# B&R Automation Studio project PloterCNC
Automation Studio 4.7.5.60 SP; technology packages: mapp 5.14.1, mappCockpit 5.14.0, mappMotion 5.14.2, mappView 5.14.2

## Configuration Config1

CPU X20CP1684, AutomationRuntime D4.73, Build 4.1.2, Safety 0.0, Vc V4.72.0

### Task classes (Cpu.sw)
```
Cyclic#1 (cycle 4000 us, tolerance 0 us):
  Initiation <- Programs.CNC_Programs.InitiationandHoming.prg
  ManualCont <- Programs.CNC_Programs.ManualContr.prg
  RuchZGCode <- Programs.CNC_Programs.RuchZGCode.prg
  live_draw <- Programs.live_drawing.live_draw.prg
Cyclic#3 (cycle 48000 us, tolerance 48000 us):
  UsrMgmtP <- Programs.UsrMgmtP.prg
Cyclic#4:
  svg_to_gco <- Programs.live_drawing.svg_to_gcode.prg
  Alarm <- Programs.Alarm.prg
Cyclic#8 (cycle 8000 us, tolerance 32000 us):
  Recipe <- Programs.Recipe.prg
DataObjects: McAcpSys
NcDataObjects: InitCncPro
Binaries: udbdef, arsvcreg, FWRules, McAcpDrv, McMechSys, mvLoader, McAcpSim, TCData, arflatprv, arcoal, TCLang, mCoWebSc, iomap, Config_4, asfw, Config_3, Role, ashwd, User, Config_1, Config_2, arconfig, Hierarchy, sysconf, ashwac, Config_6, UsrMgmt, UsrLog, TC, AlarmGnrl, Recipe_cfg, GroupGlobl, GroupFile, AlarmGlobl, GroupCnc, AlarmCnc, GroupGnrl, History, AlarmFile, Settings, Config_5, Config
Libraries: McBase, MpCnc, McAxGroup, McPathGen, McAxis, McProgInt, McAcpAx, MpAlarmX, astime, runtime, MpUserX, FileIO, MpFile, MpServer, asstring, CoTrace, AsZip, MpCom, MpBase, standard, MpWebXs, AsArSdm, MpAxis, AsBrStr, MpRecipe, sys_lib, arcert, aseth, ashw, arssl, powerlnk, asieccon, asmem, asarprof, dataobj, brsystem, asarlog, aruser, asusb, asepl, MpTweet
```

### Hardware
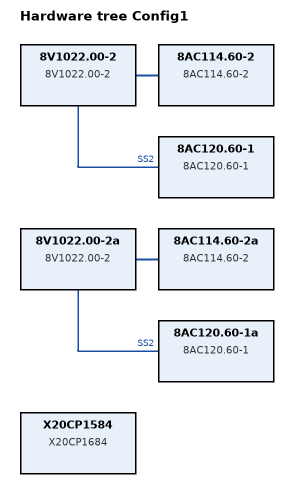
```
8AC114.60-2 : 8AC114.60-2 v1.0.0.8  [SS -> 8V1022.00-2.SS1; PLK2 -> 8AC114.60-2a.PLK2 [Cable Type=PowerlinkCable, Length=10, Version=1.0.0.2]]
8AC114.60-2a : 8AC114.60-2 v1.0.0.8  [SS -> 8V1022.00-2a.SS1; PLK1 -> X20CP1584.IF3 [Cable Type=PowerlinkCable, Length=10, Version=1.0.0.2]; PLK2 -> 8AC114.60-2.PLK2 [Cable Type=PowerlinkCable, Length=10, Version=1.0.0.2]]
8AC120.60-1 : 8AC120.60-1 v2.2.0.0  [SS -> 8V1022.00-2.SS2]
  PlugInType = Encoder
  McAcoposTypeID = AcoposPlugInConfig
8AC120.60-1a : 8AC120.60-1 v2.2.0.0  [SS -> 8V1022.00-2a.SS2]
  PlugInType = Encoder
  McAcoposTypeID = AcoposPlugInConfig
8V1022.00-2 : 8V1022.00-2 v2.2.0.0
  DriveConfiguration/Module:
    McAcoposTypeID = AcoposConfig
    ActivateACOPOSSimulationOnPLC = 0
  DriveConfiguration/Channel[1]/RealAxis:
    AxisReference = gAxisQZ
  DriveConfiguration/Channel[1]/RealAxis/MechanicalElements/Gearbox:
    InputIsReadOnly = 0
    Input = 1
    OutputIsReadOnly = 0
    Output = 1
  DriveConfiguration/Channel[1]/RealAxis/MechanicalElements/RotaryToLinearTransformation:
    ReferenceDistanceIsReadOnly = 0
    ReferenceDistance = 1.385
  DriveConfiguration/Channel[1]/RealAxis/Controller:
    ModeIsReadOnly = 0
    Mode = PositionController
  DriveConfiguration/Channel[1]/RealAxis/Controller/Mode/Position:
    ProportionalGain = 540.999939
    IntegrationTime = 0.0
    PredictionTime = 0.0004
    TotalDelayTime = 0.0004
  DriveConfiguration/Channel[1]/RealAxis/Controller/Mode/Speed:
    ProportionalGainIsReadOnly = 0
    ProportionalGain = 0.950000
    IntegrationTimeIsReadOnly = 0
    IntegrationTime = 0.0
    FilterTimeIsReadOnly = 0
    FilterTime = 0.0
  DriveConfiguration/Channel[1]/RealAxis/Controller/Mode/LoopFilters:
    LoopFilter1 = NotUsed
    LoopFilter2 = NotUsed
    LoopFilter3 = NotUsed
  DriveConfiguration/Channel[1]/RealAxis/Homing:
    Mode = Absolute
  DriveConfiguration/Channel[1]/RealAxis/Homing/Mode:
    Position = -1352
  DriveConfiguration/Channel[1]/RealAxis/Homing:
    RestorePositionVariable = 
  DriveConfiguration/Channel[1]/RealAxis/StopReaction:
    Quickstop = DecelerationLimit
    DriveError = DecelerationLimit
  DriveConfiguration/Channel[1]/RealAxis/MovementErrorLimits:
    PositionError = 1.0
    VelocityErrorMonitoring = Automatic1
  DriveConfiguration/Channel[1]/RealAxis:
    JerkFilter = NotUsed
  DriveConfiguration/Channel[1]/RealAxis/DigitalInputs/HomingSwitch:
    Level = High
  DriveConfiguration/Channel[1]/RealAxis/DigitalInputs/PositiveLimitSwitch:
    Level = Low
  DriveConfiguration/Channel[1]/RealAxis/DigitalInputs/NegativeLimitSwitch:
    Level = Low
  DriveConfiguration/Channel[1]/RealAxis/DigitalInputs/Trigger1:
    Level = High
  DriveConfiguration/Channel[1]/RealAxis/DigitalInputs/Trigger2:
    Level = High
  DriveConfiguration/Channel[1]/RealAxis/DigitalInputs/Quickstop:
    Input = Trigger2
  DriveConfiguration/Channel[1]/RealAxis/Simulation:
    SimulationModeOnPLC = SetValueGeneration
    SimulationModeOnACOPOS = NotUsed
8V1022.00-2a : 8V1022.00-2 v2.2.0.0
  DriveConfiguration/Module:
    McAcoposTypeID = AcoposConfig
    ActivateACOPOSSimulationOnPLC = 0
  DriveConfiguration/Channel[1]/RealAxis:
    AxisReference = gAxisQX
  DriveConfiguration/Channel[1]/RealAxis/MechanicalElements/Gearbox:
    InputIsReadOnly = 0
    Input = 1
    OutputIsReadOnly = 0
    Output = 1
  DriveConfiguration/Channel[1]/RealAxis/MechanicalElements/RotaryToLinearTransformation:
    ReferenceDistanceIsReadOnly = 0
    ReferenceDistance = 1.385
  DriveConfiguration/Channel[1]/RealAxis/Controller:
    ModeIsReadOnly = 0
    Mode = PositionController
  DriveConfiguration/Channel[1]/RealAxis/Controller/Mode/Position:
    ProportionalGain = 398.999969
    IntegrationTime = 0.0
    PredictionTime = 0.0004
    TotalDelayTime = 0.0004
  DriveConfiguration/Channel[1]/RealAxis/Controller/Mode/Speed:
    ProportionalGainIsReadOnly = 0
    ProportionalGain = 0.450000
    IntegrationTimeIsReadOnly = 0
    IntegrationTime = 0.0
    FilterTimeIsReadOnly = 0
    FilterTime = 0.0
  DriveConfiguration/Channel[1]/RealAxis/Controller/Mode/LoopFilters:
    LoopFilter1 = NotUsed
    LoopFilter2 = NotUsed
    LoopFilter3 = NotUsed
  DriveConfiguration/Channel[1]/RealAxis/Homing:
    Mode = Absolute
  DriveConfiguration/Channel[1]/RealAxis/Homing/Mode:
    Position = -220
  DriveConfiguration/Channel[1]/RealAxis/Homing:
    RestorePositionVariable = 
  DriveConfiguration/Channel[1]/RealAxis/StopReaction:
    Quickstop = DecelerationLimit
    DriveError = DecelerationLimit
  DriveConfiguration/Channel[1]/RealAxis/MovementErrorLimits:
    PositionError = 1.0
    VelocityErrorMonitoring = Automatic1
  DriveConfiguration/Channel[1]/RealAxis:
    JerkFilter = NotUsed
  DriveConfiguration/Channel[1]/RealAxis/DigitalInputs/HomingSwitch:
    Level = High
  DriveConfiguration/Channel[1]/RealAxis/DigitalInputs/PositiveLimitSwitch:
    Level = Low
  DriveConfiguration/Channel[1]/RealAxis/DigitalInputs/NegativeLimitSwitch:
    Level = Low
  DriveConfiguration/Channel[1]/RealAxis/DigitalInputs/Trigger1:
    Level = High
  DriveConfiguration/Channel[1]/RealAxis/DigitalInputs/Trigger2:
    Level = High
  DriveConfiguration/Channel[1]/RealAxis/DigitalInputs/Quickstop:
    Input = Trigger2
  DriveConfiguration/Channel[1]/RealAxis/Simulation:
    SimulationModeOnPLC = SetValueGeneration
    SimulationModeOnACOPOS = NotUsed
X20CP1584 : X20CP1684 v1.4.0.0
  Connector IF2:
    ActivateDevice = 1
    Mode = Manual
    InternetAddress = 192.168.0.103
    SubnetMask = 255.255.255.0
  Connector IF3:
    CycleTime = 4000
    Channel1
    ChannelID1 = McAcpBroadcast
    ChannelType1 = OCTET[24]
    InaNodeNumber = 0
  ConfigurationID = PloterCNCtat_Config1
  UserPartitionSize = 50
  VolatileGlobalPvSize = 650000
  TimerDeviceType = EPLX2X
  TimerDevice = X20CP1584.IF3
  TaskClassIdleTime = 8000
  Cyclic1Duration = 4000
  Cyclic1Tolerance = 0
  Cyclic3Duration = 48000
  Cyclic3Tolerance = 48000
  Cyclic8Duration = 8000
  Cyclic8Tolerance = 32000
  FileDevice1
  FileDeviceName1 = CNC_PrgDir
  FileDevicePath1 = F:\BrAutomation
  FileDevice2
  FileDeviceName2 = CF
  FileDevicePath2 = F:\CF
  FtpUser1
  FtpUsername1 = administrator
  FtpUserPassword1 = l2ZMc+fWbTiPJddINgK1Z9mRlNrixRAgt7akyTqvwNY=  // admin
  FtpUserSalt1 = qUW8Aw1E
  FTPAccessRight1 = 0
  ActivateDtmServer = 1
  ActivateOpcUa = 1
  OpcUaInformationModels_PV_Version = 1
```

### Config_1.axesgroup - X20CP1584/mappMotion/2AxesCNCXZ/Config_1.axesgroup
```
Element gCncXZ (Type=axesgroup)
  Type = PathGenAxesGroup
    ProcessingTaskClass = 1
    License = 1
    PhysicalAxes:
      JointAxes:
        JointAxis[1]:
          Name = QX
          AxisRef = gAxisQX
        JointAxis[2]:
          Name = QZ
          AxisRef = gAxisQZ
    MechanicalSystem:
      MechSysRef = MechSys_2AxCNCXZ
    BasicSettings:
      ModalDataBehaviour = ResetToDefault
      GeometryPlanning:
        RoundingMode = Standard
        MaxCornerDeviation = 0.0
        MaxTangentialTransitionDeviation = 0.0
        MaxRadiusDeviation = 0.001
        WorkingPlane = ZX
      TrajectoryPlanning = Basic
        LimitCheckResolution = UserDefinedTime
          Time = 0.01
        BufferTime = UserDefinedTime
          Time = 0.1
    AxesGroupFeatures:
      FeatureRef[1] = Feature_Programs
      FeatureRef[2] = Feature_Jogging
      FeatureRef[3] = Feature_MFunctions
  Alarms = MpAlarmX
```

### Config_5.axesgroupfeature - X20CP1584/mappMotion/Config_5.axesgroupfeature
```
Element Feature_MFunctions (Type=axesgroupfeature)
  Type = MFunctions
    ModalDataBehaviour = UseAxesGroupSettings
    MFunction[1]:
      IndexType = Single
        Index = 50
      Blocking = Enabled
      Output = Before
      InSimulation = NotUsed
      PvMapping = ::RuchZGCode:toolUp
      Counter
    MFunction[2]:
      IndexType = Single
        Index = 60
      Blocking = Enabled
      Output = Before
      InSimulation = NotUsed
      PvMapping = ::RuchZGCode:toolDown
      Counter
```

### GroupFile.mpcomgroup - X20CP1584/mappServices/AlarmFile/GroupFile.mpcomgroup
```
Element GroupFile (Type=mpcomgroup)
  Linking:
    Subnodes:
      0 = gAlarmXFile
  Alarms = MpAlarmX
```

### GroupGnrl.mpcomgroup - X20CP1584/mappServices/AlarmGeneral/GroupGnrl.mpcomgroup
```
Element GroupGeneral (Type=mpcomgroup)
  Linking:
    Subnodes:
      0 = gAlarmXGeneral
  Alarms = MpAlarmX
```

### AlarmGlobl.mpalarmxcore - X20CP1584/mappServices/AlarmGlobl.mpalarmxcore
```
Element gAlarmXCoreGlobal (Type=mpalarmxcore)
```

### Config_6.mpfilemanager - X20CP1584/mappServices/Config_6.mpfilemanager
```
Element FileManagement (Type=mpfilemanager)
  FileManager:
    USB = 1
    Devices:
      0:
        DeviceName = CNC_PrgDir
        Text = CNC_files
    Access:
      0:
        Folder = *
        Roles:
          0:
            Role = Everyone
            Rights:
              Visible = TRUE
              FolderRead = TRUE
              FileRead = TRUE
              FileEdit = TRUE
              FolderEdit = TRUE
  FileManagerRestrict:
    0:
      Functionality = CNCEditor
```

### GroupGlobl.mpcomgroup - X20CP1584/mappServices/GroupGlobl.mpcomgroup
```
Element GroupGlobal (Type=mpcomgroup)
  Linking:
    Subnodes:
      0 = GroupGeneral
      1 = GroupCnc
      2 = GroupFile
  Alarms = MpAlarmX
```

### History.mpalarmxhistory - X20CP1584/mappServices/History.mpalarmxhistory
```
Element gAlarmXHistory (Type=mpalarmxhistory)
```

### UsrMgmt.mpuserx - X20CP1584/mappServices/UsersConfig/UsrMgmt.mpuserx
```
Element UserMgmtX (Type=mpuserx)
  Mgr:
    PasswordLength = 4
  ServerSettings:
    Server:
      AdditionalUserData:
        [0] = mail
        [1] = telephoneNumber
  Users:
    DefUser#1:
      id = administrator
    DefUser#2:
      id = Anonymous
    DefUser#3:
      id = operator
  Groups:
    DefGroup#1:
      id = Administrator
      level = 100
      admin = TRUE
      rights:
        [0] = FullAccess
    DefGroup#2:
      id = Everyone
      rights:
        [0] = ViewOnly
    DefGroup#3:
      id = Operator
      level = 50
      admin = TRUE
      rights:
        [0] = FullAccess
```

## Configuration Simulation

CPU X20CP1584, AutomationRuntime D4.73, Build 4.1.2, Safety 0.0, Vc V4.72.0

CPU X20CP1684, AutomationRuntime D4.73, Build 4.1.2, Safety 0.0, Vc V4.72.0

### Task classes (Cpu.sw)
```
Cyclic#1 (cycle 4000 us, tolerance 0 us):
  Initiation <- Programs.CNC_Programs.InitiationandHoming.prg
  ManualCont <- Programs.CNC_Programs.ManualContr.prg
  live_draw <- Programs.live_drawing.live_draw.prg
  RuchZGCode <- Programs.CNC_Programs.RuchZGCode.prg
  PloterCfg <- MSpltrFmu.PloterCfg.prg
Cyclic#4:
  svg_to_gco <- Programs.live_drawing.svg_to_gcode.prg
  Alarm <- Programs.Alarm.prg
Cyclic#8 (cycle 8000 us, tolerance 32000 us):
  Recipe <- Programs.Recipe.prg
DataObjects: McAcpSys
NcDataObjects: InitCncPro
Binaries: udbdef, arsvcreg, FWRules, McAcpDrv, McMechSys, mvLoader, McAcpSim, TCData, arflatprv, arcoal, TCLang, mCoWebSc, iomap, Config_4, asfw, Config_3, Role, ashwd, User, Config_1, Config_2, arconfig, Hierarchy, sysconf, ashwac, Config_6, UsrMgmt, UsrLog, TC, AlarmGnrl, Recipe_cfg, GroupGlobl, GroupFile, AlarmGlobl, GroupCnc, AlarmCnc, GroupGnrl, History, AlarmFile, Settings, Config_5, Config
Libraries: McBase, MpCnc, McAxGroup, McPathGen, McAxis, McProgInt, McAcpAx, MpAlarmX, astime, runtime, MpUserX, FileIO, MpFile, MpServer, asstring, CoTrace, AsZip, MpCom, MpBase, standard, MpWebXs, AsArSdm, MpAxis, AsBrStr, MpRecipe, sys_lib, MpTweet, MSpltrLib, arcert, aseth, ashw, arssl, powerlnk, asieccon, asmem, asarprof, dataobj, asarlog, aruser, asusb, asepl, dvframe, CNC_FMULib, brsystem
```

### Task classes (Cpu.sw)
```
Cyclic#1 (cycle 4000 us, tolerance 0 us):
  Initiation <- CNC_Programs.InitiationandHoming.prg
  ManualCont <- CNC_Programs.ManualContr.prg
  live_draw <- live_drawing.live_draw.prg
  RuchZGCode <- RuchZGCode.prg
Cyclic#3 (cycle 48000 us, tolerance 48000 us):
  UsrMgmtP <- UserManagement.UsrMgmtP.prg
Cyclic#4:
  svg_to_gco <- live_drawing.svg_to_gcode.prg
  Alarm <- Alarm.prg
Cyclic#8 (cycle 8000 us, tolerance 32000 us):
  Recipe <- Recipe.prg
DataObjects: McAcpSys
NcDataObjects: InitCncPro
Binaries: udbdef, arsvcreg, FWRules, McAcpDrv, McMechSys, mvLoader, McAcpSim, TCData, arflatprv, arcoal, TCLang, mCoWebSc, iomap, Config_4, asfw, Config_3, Role, ashwd, User, Config_1, Config_2, arconfig, Hierarchy, sysconf, ashwac, Config_6, UsrMgmt, UsrLog, TC, AlarmGnrl, Recipe_cfg, GroupGlobl, GroupFile, AlarmGlobl, GroupCnc, AlarmCnc, GroupGnrl, History, AlarmFile, Settings, Config_5, Config
Libraries: McBase, MpCnc, McAxGroup, McPathGen, McAxis, McProgInt, McAcpAx, MpAlarmX, astime, runtime, MpUserX, FileIO, MpFile, MpServer, asstring, CoTrace, AsZip, MpCom, MpBase, standard, MpWebXs, AsArSdm, MpAxis, AsBrStr, MpRecipe, sys_lib, arcert, aseth, ashw, arssl, powerlnk, asieccon, asmem, asarprof, dataobj, brsystem, asarlog, aruser, asusb, asepl, CNC_FMULib
```

### Hardware
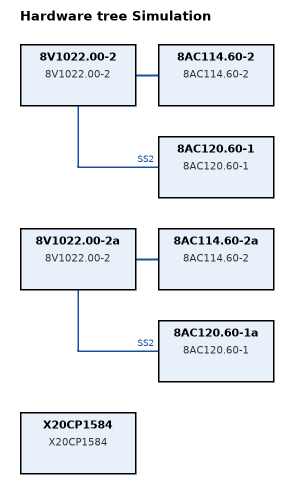
```
8AC114.60-2 : 8AC114.60-2 v1.0.0.8  [SS -> 8V1022.00-2.SS1; PLK2 -> 8AC114.60-2a.PLK2 [Cable Type=PowerlinkCable, Length=10, Version=1.0.0.2]]
8AC114.60-2a : 8AC114.60-2 v1.0.0.8  [SS -> 8V1022.00-2a.SS1; PLK1 -> X20CP1584.IF3 [Cable Type=PowerlinkCable, Length=10, Version=1.0.0.2]; PLK2 -> 8AC114.60-2.PLK2 [Cable Type=PowerlinkCable, Length=10, Version=1.0.0.2]]
8AC120.60-1 : 8AC120.60-1 v2.2.0.0  [SS -> 8V1022.00-2.SS2]
  PlugInType = Encoder
  McAcoposTypeID = AcoposPlugInConfig
8AC120.60-1a : 8AC120.60-1 v2.2.0.0  [SS -> 8V1022.00-2a.SS2]
  PlugInType = Encoder
  McAcoposTypeID = AcoposPlugInConfig
8V1022.00-2 : 8V1022.00-2 v2.2.0.0
  DriveConfiguration/Module:
    McAcoposTypeID = AcoposConfig
    ActivateACOPOSSimulationOnPLC = 0
  DriveConfiguration/Channel[1]/RealAxis:
    AxisReference = gAxisQZ
  DriveConfiguration/Channel[1]/RealAxis/MechanicalElements/Gearbox:
    InputIsReadOnly = 0
    Input = 1
    OutputIsReadOnly = 0
    Output = 1
  DriveConfiguration/Channel[1]/RealAxis/MechanicalElements/RotaryToLinearTransformation:
    ReferenceDistanceIsReadOnly = 0
    ReferenceDistance = 1.385
  DriveConfiguration/Channel[1]/RealAxis/Controller:
    ModeIsReadOnly = 0
    Mode = PositionController
  DriveConfiguration/Channel[1]/RealAxis/Controller/Mode/Position:
    ProportionalGain = 540.999939
    IntegrationTime = 0.0
    PredictionTime = 0.0004
    TotalDelayTime = 0.0004
  DriveConfiguration/Channel[1]/RealAxis/Controller/Mode/Speed:
    ProportionalGainIsReadOnly = 0
    ProportionalGain = 0.950000
    IntegrationTimeIsReadOnly = 0
    IntegrationTime = 0.0
    FilterTimeIsReadOnly = 0
    FilterTime = 0.0
  DriveConfiguration/Channel[1]/RealAxis/Controller/Mode/LoopFilters:
    LoopFilter1 = NotUsed
    LoopFilter2 = NotUsed
    LoopFilter3 = NotUsed
  DriveConfiguration/Channel[1]/RealAxis/Homing:
    Mode = Absolute
  DriveConfiguration/Channel[1]/RealAxis/Homing/Mode:
    Position = 0
  DriveConfiguration/Channel[1]/RealAxis/Homing:
    RestorePositionVariable = 
  DriveConfiguration/Channel[1]/RealAxis/StopReaction:
    Quickstop = DecelerationLimit
    DriveError = DecelerationLimit
  DriveConfiguration/Channel[1]/RealAxis/MovementErrorLimits:
    PositionError = 1.0
    VelocityErrorMonitoring = Automatic1
  DriveConfiguration/Channel[1]/RealAxis:
    JerkFilter = NotUsed
  DriveConfiguration/Channel[1]/RealAxis/DigitalInputs/HomingSwitch:
    Level = High
  DriveConfiguration/Channel[1]/RealAxis/DigitalInputs/PositiveLimitSwitch:
    Level = Low
  DriveConfiguration/Channel[1]/RealAxis/DigitalInputs/NegativeLimitSwitch:
    Level = Low
  DriveConfiguration/Channel[1]/RealAxis/DigitalInputs/Trigger1:
    Level = High
  DriveConfiguration/Channel[1]/RealAxis/DigitalInputs/Trigger2:
    Level = High
  DriveConfiguration/Channel[1]/RealAxis/DigitalInputs/Quickstop:
    Input = Trigger2
  DriveConfiguration/Channel[1]/RealAxis/Simulation:
    SimulationModeOnPLC = SetValueGeneration
    SimulationModeOnACOPOS = NotUsed
8V1022.00-2a : 8V1022.00-2 v2.2.0.0
  DriveConfiguration/Module:
    McAcoposTypeID = AcoposConfig
    ActivateACOPOSSimulationOnPLC = 0
  DriveConfiguration/Channel[1]/RealAxis:
    AxisReference = gAxisQX
  DriveConfiguration/Channel[1]/RealAxis/MechanicalElements/Gearbox:
    InputIsReadOnly = 0
    Input = 1
    OutputIsReadOnly = 0
    Output = 1
  DriveConfiguration/Channel[1]/RealAxis/MechanicalElements/RotaryToLinearTransformation:
    ReferenceDistanceIsReadOnly = 0
    ReferenceDistance = 1.385
  DriveConfiguration/Channel[1]/RealAxis/Controller:
    ModeIsReadOnly = 0
    Mode = PositionController
  DriveConfiguration/Channel[1]/RealAxis/Controller/Mode/Position:
    ProportionalGain = 398.999969
    IntegrationTime = 0.0
    PredictionTime = 0.0004
    TotalDelayTime = 0.0004
  DriveConfiguration/Channel[1]/RealAxis/Controller/Mode/Speed:
    ProportionalGainIsReadOnly = 0
    ProportionalGain = 0.450000
    IntegrationTimeIsReadOnly = 0
    IntegrationTime = 0.0
    FilterTimeIsReadOnly = 0
    FilterTime = 0.0
  DriveConfiguration/Channel[1]/RealAxis/Controller/Mode/LoopFilters:
    LoopFilter1 = NotUsed
    LoopFilter2 = NotUsed
    LoopFilter3 = NotUsed
  DriveConfiguration/Channel[1]/RealAxis/Homing:
    Mode = Absolute
  DriveConfiguration/Channel[1]/RealAxis/Homing/Mode:
    Position = 0
  DriveConfiguration/Channel[1]/RealAxis/Homing:
    RestorePositionVariable = 
  DriveConfiguration/Channel[1]/RealAxis/StopReaction:
    Quickstop = DecelerationLimit
    DriveError = DecelerationLimit
  DriveConfiguration/Channel[1]/RealAxis/MovementErrorLimits:
    PositionError = 1.0
    VelocityErrorMonitoring = Automatic1
  DriveConfiguration/Channel[1]/RealAxis:
    JerkFilter = NotUsed
  DriveConfiguration/Channel[1]/RealAxis/DigitalInputs/HomingSwitch:
    Level = High
  DriveConfiguration/Channel[1]/RealAxis/DigitalInputs/PositiveLimitSwitch:
    Level = Low
  DriveConfiguration/Channel[1]/RealAxis/DigitalInputs/NegativeLimitSwitch:
    Level = Low
  DriveConfiguration/Channel[1]/RealAxis/DigitalInputs/Trigger1:
    Level = High
  DriveConfiguration/Channel[1]/RealAxis/DigitalInputs/Trigger2:
    Level = High
  DriveConfiguration/Channel[1]/RealAxis/DigitalInputs/Quickstop:
    Input = Trigger2
  DriveConfiguration/Channel[1]/RealAxis/Simulation:
    SimulationModeOnPLC = SetValueGeneration
    SimulationModeOnACOPOS = NotUsed
X20CP1584 : X20CP1584 v1.6.0.0
  Connector IF2:
    ActivateDevice = 1
    Mode = Manual
    InternetAddress = 192.168.0.103
    SubnetMask = 255.255.255.0
    Vnc1
    VncKeyMappingFile1 = VC\PS2-Keyboard.dis
  Connector IF3:
    CycleTime = 4000
    Channel1
    ChannelID1 = McAcpBroadcast
    ChannelType1 = OCTET[24]
    InaNodeNumber = 0
  ConfigurationID = PloterCNCtat_Config1
  UserPartitionSize = 50
  Simulation = 1
  VolatileGlobalPvSize = 650000
  TimerDeviceType = EPLX2X
  TimerDevice = X20CP1584.IF3
  TaskClassIdleTime = 8000
  Cyclic1Duration = 4000
  Cyclic1Tolerance = 0
  Cyclic3Duration = 48000
  Cyclic3Tolerance = 48000
  Cyclic8Duration = 8000
  Cyclic8Tolerance = 32000
  FileDevice1
  FileDeviceName1 = CNC_PrgDir
  FileDevicePath1 = C:\BrAutomation
  FileDevice2
  FileDeviceName2 = CF
  FileDevicePath2 = C:\CF
  FtpUser1
  FtpUsername1 = administrator
  FtpUserPassword1 = l2ZMc+fWbTiPJddINgK1Z9mRlNrixRAgt7akyTqvwNY=  // admin
  FtpUserSalt1 = qUW8Aw1E
  FTPAccessRight1 = 0
  ActivateDtmServer = 1
  ActivateOpcUa = 1
  OpcUaInformationModels_PV_Version = 1
```

### AlarmCnc.mpalarmxcore - X20CP1584/mappServices/AlarmCnc/AlarmCnc.mpalarmxcore
```
Element gAlarmXCnc (Type=mpalarmxcore)
  mapp.AlarmX.Core.Configuration:
    [0]:
      Name = AxisXOver
      Message = Axis X over preprogrammed area
      Code = 2
      Behavior = LevelMonitoring
        Monitoring:
          MonitoredPV = ::gParameter.limit_X_pos
          LowLimitEnable = Static
          HighLimitEnable = Static
            Limit = 521
    [1]:
      Name = AxisZOver
      Message = Axis Z over preprogrammed area
      Code = 3
      Behavior = LevelMonitoring
        Monitoring:
          MonitoredPV = ::gParameter.limit_Z_pos
          LowLimitEnable = Static
          HighLimitEnable = Static
            Limit = 421
    [2]:
      Name = VelocityLimitX
      Message = Current velocity of axis X is higher then limit
      Code = 7
      Behavior = LevelMonitoring
        Monitoring:
          MonitoredPV = ::gParameter.set_X_vel
          HighLimitEnable = Dynamic
            LimitPV = ::gParameter.limit_vel
    [3]:
      Name = VelocityLimitY
      Message = Current velocity of axis Y is higher then limit
      Code = 8
      Behavior = LevelMonitoring
        Monitoring:
          MonitoredPV = ::gParameter.set_Z_vel
          HighLimitEnable = Dynamic
            LimitPV = ::gParameter.limit_vel
```

### AlarmFile.mpalarmxcore - X20CP1584/mappServices/AlarmFile/AlarmFile.mpalarmxcore
```
Element gAlarmXFile (Type=mpalarmxcore)
  mapp.AlarmX.Core.Configuration:
    [0]:
      Name = MotionPadError
      Code = 4
      Behavior = LevelMonitoring
        Monitoring:
          MonitoredPV = ::gMotionPadError
          LowLimitEnable = Static
          HighLimitEnable = Static
    [1]:
      Name = FileNotSaved
      Code = 5
    [2]:
      Name = USBConnectionFailure
      Message = USB Connection Failure
      Code = 100
    [3]:
      Name = FTPServerNotConnected
      Message = FTP server not connected
      Code = 101
      Behavior = PersistentAlarm
    [4]:
      Name = FTPServerDisconnected
      Message = FTP server disconnected
      Code = 102
    [5]:
      Name = FOpenAlarm
      Message = Error in opening file
      Code = 104
    [6]:
      Name = FCreateAlarm
      Message = Error in creation of new file
      Severity = 105
    [7]:
      Name = FCloseAlarm
      Message = Error in closing the file
      Severity = 107
    [8]:
      Name = FWriteAlarm
      Message = Error in writing to the file
      Severity = 108
```

### AlarmGnrl.mpalarmxcore - X20CP1584/mappServices/AlarmGeneral/AlarmGnrl.mpalarmxcore
```
Element gAlarmXGeneral (Type=mpalarmxcore)
  mapp.AlarmX.Core.Configuration:
    [0]:
      Name = EmergencyStop
      Code = 1
      Behavior = PersistentAlarm
    [1]:
      Name = RecipeAlarm
      Message = Error in creation of recipe
      Behavior = DiscreteValueMonitoring
        Monitoring:
          MonitoredPV = ::Recipe:MpRecipeUI_0.Error
          TriggerValues:
            [0] = true
```

### Config.mpfilemanager - X20CP1584/mappServices/Config.mpfilemanager
```
Element FileManagement (Type=mpfilemanager)
```

### Config_6.mpfilemanager - X20CP1584/mappServices/Config_6.mpfilemanager
```
Element FileManagement (Type=mpfilemanager)
  FileManager:
    USB = 1
    Devices:
      0:
        DeviceName = CNC_PrgDir
        Text = CNC_files
    Access:
      0:
        Folder = *
        Roles:
          0:
            Role = Administrator
            Rights:
              Visible = TRUE
              FolderRead = TRUE
              FileRead = TRUE
              FileEdit = TRUE
              FolderEdit = TRUE
          1:
            Role = Operator
            Rights:
              Visible = TRUE
              FolderRead = TRUE
              FileRead = TRUE
              FileEdit = TRUE
              FolderEdit = TRUE
  FileManagerRestrict:
    0:
      Functionality = CNCEditor
```

### Recipe_cfg.mprecipexml - X20CP1584/mappServices/Recipe_cfg.mprecipexml
```
Element gRecipeXml (Type=mprecipexml)
  Alarms = MpAlarmX
```

### Config_2.axis - X20CP1684/mappMotion/2AxesCNCXZ/Config_2.axis
```
Element gAxisQX (Type=axis)
  BaseTypeIsReadOnly = 0
  BaseType = LinearBounded
    MeasurementUnit = 5066068
    MeasurementResolutionIsReadOnly = 0
    MeasurementResolution = 0.01
    CountDirectionIsReadOnly = 0
    CountDirection = Standard
  MovementLimitsIsReadOnly = 0
  MovementLimits = Internal
    Position:
      LowerLimitMin = -1.79769313486231E308
      UpperLimitMax = 1.79769313486231E308
      LowerLimit = -2
      UpperLimit = 522
    VelocityIsReadOnly = 0
    Velocity:
      VelocityMax = 3.4E38
      Velocity = 100
    AccelerationIsReadOnly = 0
    Acceleration:
      AccelerationMax = 3.4E38
      Acceleration = 1000
    DecelerationIsReadOnly = 0
    Deceleration:
      DecelerationMax = 3.4E38
      Deceleration = 1000
  Alarms = MpAlarmX
Element gAxisQZ (Type=axis)
  BaseTypeIsReadOnly = 0
  BaseType = LinearBounded
    MeasurementUnit = 5066068
    MeasurementResolutionIsReadOnly = 0
    MeasurementResolution = 0.01
    CountDirectionIsReadOnly = 0
    CountDirection = Standard
  MovementLimitsIsReadOnly = 0
  MovementLimits = Internal
    Position:
      LowerLimitMin = -1.79769313486231E308
      UpperLimitMax = 1.79769313486231E308
      LowerLimit = -2
      UpperLimit = 422
    VelocityIsReadOnly = 0
    Velocity:
      VelocityMax = 3.4E38
      Velocity = 100
    AccelerationIsReadOnly = 0
    Acceleration:
      AccelerationMax = 3.4E38
      Acceleration = 1000
    DecelerationIsReadOnly = 0
    Deceleration:
      DecelerationMax = 3.4E38
      Deceleration = 1000
  Alarms = MpAlarmX
```

### Config_3.mechanicalsystem - X20CP1684/mappMotion/2AxesCNCXZ/Config_3.mechanicalsystem
```
Element MechSys_2AxCNCXZ (Type=mechanicalsystem)
  Type = 2AxesCNC
    Subtype = 2AxesCNCXZ
      CoordinatesNames = Default
        XCoordinateName = X
        ZCoordinateName = Z
      WireFrameModel = Standard
        FlangeToTcp = ConnectionLine
          Distance = 0.0
      JointAxesPositionLimits:
        JointAxis[1] = UseAxisLimits
        JointAxis[2] = UseAxisLimits
```

### Config_4.axesgroupfeature - X20CP1684/mappMotion/2AxesCNCXZ/Config_4.axesgroupfeature
```
Element Feature_Programs (Type=axesgroupfeature)
  Type = Program
    ModalDataBehaviour = UseAxesGroupSettings
    InitialSettings:
      InterpolationTypes = LinearRapid
      PositionCoordinates = Absolute
      CircleCoordinates = Relative
      JACS_ACSProgramming = JACS
      ContourConnection = Inactive
      ProgrammingUnits = UseAxesGroupSettings
      Feedrates:
        FeedCharacteristic = StandardCharacteristic
        FeedType = Feedrate
        FeedReduction = Inactive
        FeedrateValue = 0.0
        InverseFeedrateValue = 0.0
        FeedratePerRevValue = 0.0
    DefaultLanguage = BRGCode
    Location = Default
      FileDevice = CNC_PrgDir
Element Feature_Jogging (Type=axesgroupfeature)
  Type = Jogging
Element Feature_Programs_1 (Type=axesgroupfeature)
  Type = Program
    ModalDataBehaviour = UseAxesGroupSettings
    InitialSettings:
      InterpolationTypes = LinearRapid
      PositionCoordinates = Absolute
      CircleCoordinates = Relative
      JACS_ACSProgramming = JACS
      ContourConnection = Inactive
      ProgrammingUnits = UseAxesGroupSettings
      Feedrates:
        FeedCharacteristic = StandardCharacteristic
        FeedType = Feedrate
        FeedReduction = Inactive
        FeedrateValue = 0.0
        InverseFeedrateValue = 0.0
        FeedratePerRevValue = 0.0
    DefaultLanguage = BRGCode
    Location = Default
      FileDevice = CNC_PrgDir
Element Feature_Programs_2 (Type=axesgroupfeature)
  Type = Program
    ModalDataBehaviour = UseAxesGroupSettings
    InitialSettings:
      InterpolationTypes = LinearRapid
      PositionCoordinates = Absolute
      CircleCoordinates = Relative
      JACS_ACSProgramming = JACS
      ContourConnection = Inactive
      ProgrammingUnits = UseAxesGroupSettings
      Feedrates:
        FeedCharacteristic = StandardCharacteristic
        FeedType = Feedrate
        FeedReduction = Inactive
        FeedrateValue = 0.0
        InverseFeedrateValue = 0.0
        FeedratePerRevValue = 0.0
    DefaultLanguage = BRGCode
    Location = Default
      FileDevice = CNC_PrgDir
```

### GroupCnc.mpcomgroup - X20CP1684/mappServices/AlarmCnc/GroupCnc.mpcomgroup
```
Element GroupCnc (Type=mpcomgroup)
  Linking:
    Subnodes:
      0 = gAlarmXCnc
  Alarms = MpAlarmX
```

### Config_6.mpfilemanager - X20CP1684/mappServices/Config_6.mpfilemanager
```
Element FileManagement (Type=mpfilemanager)
  FileManager:
    USB = 1
    Devices:
      0:
        DeviceName = CNC_PrgDir
        Text = CNC_files
    Access:
      0:
        Folder = *
        Roles:
          0:
            Role = 
            Rights:
              Visible = TRUE
              FolderRead = TRUE
              FileRead = TRUE
              FileEdit = TRUE
              FolderEdit = TRUE
  FileManagerRestrict:
    0:
      Functionality = CNCEditor
```

### UsrMgmt.mpuserx - X20CP1684/mappServices/UsersConfig/UsrMgmt.mpuserx
```
Element UserMgmtX (Type=mpuserx)
  Mgr:
    PasswordLength = 4
    EditSameLevel = TRUE
  ServerSettings:
    Server:
      AdditionalUserData:
        [0] = mail
        [1] = telephoneNumber
  Users:
    DefUser#1:
      id = administrator
      name = Administrator1
    DefUser#2:
      id = Anonymous
      name = Anonymous
    DefUser#3:
      id = operator
      name = Operator1
  Groups:
    DefGroup#1:
      id = Administrator
      level = 100
      admin = TRUE
      rights:
        [0] = FullAccess
    DefGroup#2:
      id = Everyone
      level = 0
      rights:
        [0] = ViewOnly
    DefGroup#3:
      id = Operator
      level = 100
      rights:
        [0] = FullAccess
```

## Logical view

Binary libraries used (declarations not repeated): operator, runtime, astime, AsIecCon, FileIO, asstring, AsZip, standard, AsArSdm, AsBrStr, sys_lib, brsystem, McBase 5.14.2, McAcpAx 5.14.2, McPathGen 5.14.2, McAxGroup 5.14.2, McAxis 5.14.2, McProgInt 5.14.2, MpCnc 5.14.2, MpAxis 5.14.2, MpBase 5.14.1, MpWebXs 5.14.1, MpRecipe 5.14.1, MpUserX 5.14.1, MpTweet 5.14.1, MpFile 5.14.1, MpAlarmX 5.14.1, MpCom 5.14.1, MpServer 5.14.1, CoTrace 5.14.0, MTBasics 2.30.2, MTTypes 1.03.4, AsSMTP

### Global.typ - Global data types
```iecst
TYPE
	SaveParameterType : 	STRUCT
		limit_X_pos : REAL := 520;
		limit_Z_pos : REAL := 420;
		limit_acc : REAL := 1000;
		limit_vel : REAL := 100;
		limit_dec : REAL := 1000;
		set_Z_vel : REAL := 100;
		set_X_vel : REAL := 100;
	END_STRUCT;
END_TYPE
```

### Global.var - Global variables
```iecst
(*Insert your comment here.*)
VAR
	Show : BOOL := FALSE;
	NumericInput : USINT := 0;
	SliderInput : USINT := 0;
	ButtonEnable : BOOL;
	CncName : STRING[80];
	CncNameCopy : STRING[80];
	CncParameters : MpCnc2AxisParType;
	CncPosX : INT;
	CncPosY : INT;
	gActiveTool : BOOL; (*TRUE-długopis pisze; FALSE- długopis nie pisze*)
	gAlarmActive : BOOL;
	gManualContr : BOOL; (*TRUE- sterowanie ręczne; FALSE-inny tryb*)
	gMoveAbsoluteX : BOOL;
	gMoveAbsoluteY : BOOL;
	gMsgBox : BOOL;
	gMsgBox2 : BOOL;
	gMsgBox3 : BOOL;
	gMsgBox4 : BOOL;
END_VAR
VAR RETAIN
	gParameter : SaveParameterType;
END_VAR
VAR
	gStartValueChanging : BOOL;
END_VAR
VAR CONSTANT
	HomingMode : McHomingModeEnum := mcHOMING_ABSOLUTE;
END_VAR
VAR
	MoveMachine : UINT;
	MpAxisBasicX : MpAxisBasic;
	MpAxisBasicY : MpAxisBasic;
	MpBasicParametersX : MpAxisBasicParType := (Homing:=(Mode:=mcHOMING_ABSOLUTE));
	MpBasicParametersY : MpAxisBasicParType := (Homing:=(Mode:=mcHOMING_ABSOLUTE));
	MpCnc2Axis_0 : MpCnc2Axis;
	gAutomaticContr : BOOL;
END_VAR
(*FMU variables*)
VAR
	MSpltr1 : MSpltr;
	gTorqueY : LREAL;
	gTorqueX : LREAL;
	gPozycjaY : LREAL;
	gPozycjaX : LREAL;
	MSpltrView_0 : MSpltrView;
END_VAR
```

### Package Logical/Libraries - Global libraries

- Visualisation Logical/mappView (not shown)

### Library Logical/MSpltrFmu/MSpltrLib (ANSIC)
Depends on: sys_lib

#### Types.typ - Exported data types
```iecst
TYPE
	MSpltrLibFmi2CbType : 	STRUCT
		Logger : UDINT;
		AllocateMemory : UDINT;
		FreeMemory : UDINT;
		StepFinished : UDINT;
		ComponentEnvironment : UDINT;
	END_STRUCT;
	MSpltrLibFmi2IfType : 	STRUCT
		Enabled : BOOL;
		StartTime : LREAL;
		EndTime : LREAL;
		CurrentTime : LREAL;
		StepSize : LREAL;
		Error : DINT;
		Instance : UDINT;
		Callbacks : MSpltrLibFmi2CbType;
	END_STRUCT;
	MSpltrInternalType : 	STRUCT
		Fmi2 : MSpltrLibFmi2IfType;
	END_STRUCT;
END_TYPE
```

#### MSpltrLib.fun - Exported functions and function blocks
```iecst
FUNCTION_BLOCK MSpltrView
	VAR_INPUT
		Enable : BOOL;
		InstRef : REFERENCE TO MSpltrInternalType;
	END_VAR
	VAR_OUTPUT
		ObjPos : ARRAY[0..18] OF REAL;
	END_VAR
	VAR
		vInternal : ARRAY[0..18] OF LREAL;
	END_VAR
END_FUNCTION_BLOCK

FUNCTION_BLOCK MSpltr (**) (*$GROUP=User,$CAT=User,$GROUPICON=User.png,$CATICON=User.png*) (*Fmu.Type="MSpltr",Fmu.ModelName="MSpltr",Fmu.GUID="{d25602c7-833a-5e8d-e356-ec0e85f22cec}",Fmu.LocalPath="C:\projects\MS_FMU\MSpltr.fmu",Fmu.Updated="2019-09-27 13:58:32"*)
	VAR_INPUT
		Enable : BOOL;
	END_VAR
	VAR_OUTPUT
		InstRef : UDINT;
	END_VAR
	VAR
		Internal : MSpltrInternalType;
	END_VAR
	VAR_INPUT
		InputX : LREAL; (*InputX*)
		InputY : LREAL; (*InputY*)
	END_VAR
	VAR_OUTPUT
		PositionX : LREAL; (*PositionX*)
		PositionY : LREAL; (*PositionY*)
		SpeedX : LREAL; (*der(P1.s)*)
		SpeedY : LREAL; (*der(P2.s)*)
		TorqueX : LREAL; (*TorqueX*)
		TorqueY : LREAL; (*TorqueY*)
	END_VAR
END_FUNCTION_BLOCK
```

#### fmi2.cpp
```cpp
/********************************************************************
 * COPYRIGHT -- B&R Industrial Automation GmbH
 ********************************************************************
 * Program: fmu
 * File: fmu.cpp
 * Author: hkellinger
 * Created: June 25, 2015
 ********************************************************************
 * Basic fmu declarations
 ********************************************************************/

#ifdef __cplusplus
unsigned long bur_heap_size = 4096000;
#endif
```

#### fmi2Functions.h
```c
#ifndef fmi2Functions_h
#define fmi2Functions_h

/* This header file must be utilized when compiling a FMU.
   It defines all functions of the
         FMI 2.0 Model Exchange and Co-Simulation Interface.

   In order to have unique function names even if several FMUs
   are compiled together (e.g. for embedded systems), every "real" function name
   is constructed by prepending the function name by "FMI2_FUNCTION_PREFIX".
   Therefore, the typical usage is:

      #define FMI2_FUNCTION_PREFIX MyModel_
      #include "fmi2Functions.h"

   As a result, a function that is defined as "fmi2GetDerivatives" in this header file,
   is actually getting the name "MyModel_fmi2GetDerivatives".

   This only holds if the FMU is shipped in C source code, or is compiled in a
   static link library. For FMUs compiled in a DLL/sharedObject, the "actual" function
   names are used and "FMI2_FUNCTION_PREFIX" must not be defined.

   Revisions:
   - Apr.  9, 2014: all prefixes "fmi" renamed to "fmi2" (decision from April 8)
   - Mar. 26, 2014: FMI_Export set to empty value if FMI_Export and FMI_FUNCTION_PREFIX
                    are not defined (#173)
   - Oct. 11, 2013: Functions of ModelExchange and CoSimulation merged:
                      fmiInstantiateModel , fmiInstantiateSlave  -> fmiInstantiate
                      fmiFreeModelInstance, fmiFreeSlaveInstance -> fmiFreeInstance
                      fmiEnterModelInitializationMode, fmiEnterSlaveInitializationMode -> fmiEnterInitializationMode
                      fmiExitModelInitializationMode , fmiExitSlaveInitializationMode  -> fmiExitInitializationMode
                      fmiTerminateModel, fmiTerminateSlave  -> fmiTerminate
                      fmiResetSlave -> fmiReset (now also for ModelExchange and not only for CoSimulation)
                    Functions renamed:
                      fmiUpdateDiscreteStates -> fmiNewDiscreteStates
   - June 13, 2013: Functions removed:
                       fmiInitializeModel
                       fmiEventUpdate
                       fmiCompletedEventIteration
                       fmiInitializeSlave
                    Functions added:
                       fmiEnterModelInitializationMode
                       fmiExitModelInitializationMode
                       fmiEnterEventMode
                       fmiUpdateDiscreteStates
                       fmiEnterContinuousTimeMode
                       fmiEnterSlaveInitializationMode;
                       fmiExitSlaveInitializationMode;
   - Feb. 17, 2013: Portability improvements:
                       o DllExport changed to FMI_Export
                       o FUNCTION_PREFIX changed to FMI_FUNCTION_PREFIX
                       o Allow undefined FMI_FUNCTION_PREFIX (meaning no prefix is used)
                    Changed function name "fmiTerminate" to "fmiTerminateModel" (due to #113)
                    Changed function name "fmiGetNominalContinuousState" to
                                          "fmiGetNominalsOfContinuousStates"
                    Removed fmiGetStateValueReferences.
   - Nov. 14, 2011: Adapted to FMI 2.0:
                       o Split into two files (fmiFunctions.h, fmiTypes.h) in order
                         that code that dynamically loads an FMU can directly
                         utilize the header files).
                       o Added C++ encapsulation of C-part, in order that the header
                         file can be directly utilized in C++ code.
                       o fmiCallbackFunctions is passed as pointer to fmiInstantiateXXX
                       o stepFinished within fmiCallbackFunctions has as first
                         argument "fmiComponentEnvironment" and not "fmiComponent".
                       o New functions to get and set the complete FMU state
                         and to compute partial derivatives.
   - Nov.  4, 2010: Adapted to specification text:
                       o fmiGetModelTypesPlatform renamed to fmiGetTypesPlatform
                       o fmiInstantiateSlave: Argument GUID     replaced by fmuGUID
                                              Argument mimetype replaced by mimeType
                       o tabs replaced by spaces
   - Oct. 16, 2010: Functions for FMI for Co-simulation added
   - Jan. 20, 2010: stateValueReferencesChanged added to struct fmiEventInfo (ticket #27)
                    (by M. Otter, DLR)
                    Added WIN32 pragma to define the struct layout (ticket #34)
                    (by J. Mauss, QTronic)
   - Jan.  4, 2010: Removed argument intermediateResults from fmiInitialize
                    Renamed macro fmiGetModelFunctionsVersion to fmiGetVersion
                    Renamed macro fmiModelFunctionsVersion to fmiVersion
                    Replaced fmiModel by fmiComponent in decl of fmiInstantiateModel
                    (by J. Mauss, QTronic)
   - Dec. 17, 2009: Changed extension "me" to "fmi" (by Martin Otter, DLR).
   - Dez. 14, 2009: Added eventInfo to meInitialize and added
                    meGetNominalContinuousStates (by Martin Otter, DLR)
   - Sept. 9, 2009: Added DllExport (according to Peter Nilsson's suggestion)
                    (by A. Junghanns, QTronic)
   - Sept. 9, 2009: Changes according to FMI-meeting on July 21:
                    meInquireModelTypesVersion     -> meGetModelTypesPlatform
                    meInquireModelFunctionsVersion -> meGetModelFunctionsVersion
                    meSetStates                    -> meSetContinuousStates
                    meGetStates                    -> meGetContinuousStates
                    removal of meInitializeModelClass
                    removal of meGetTime
                    change of arguments of meInstantiateModel
                    change of arguments of meCompletedIntegratorStep
                    (by Martin Otter, DLR):
   - July 19, 2009: Added "me" as prefix to file names (by Martin Otter, DLR).
   - March 2, 2009: Changed function definitions according to the last design
                    meeting with additional improvements (by Martin Otter, DLR).
   - Dec. 3 , 2008: First version by Martin Otter (DLR) and Hans Olsson (Dynasim).

   Copyright © 2008-2011 MODELISAR consortium,
               2012-2013 Modelica Association Project "FMI"
               All rights reserved.
   This file is licensed by the copyright holders under the BSD 2-Clause License
   (http://www.opensource.org/licenses/bsd-license.html):

   ----------------------------------------------------------------------------
   Redistribution and use in source and binary forms, with or without
   modification, are permitted provided that the following conditions are met:

   - Redistributions of source code must retain the above copyright notice,
     this list of conditions and the following disclaimer.
   - Redistributions in binary form must reproduce the above copyright notice,
     this list of conditions and the following disclaimer in the documentation
     and/or other materials provided with the distribution.
   - Neither the name of the copyright holders nor the names of its
     contributors may be used to endorse or promote products derived
     from this software without specific prior written permission.

   THIS SOFTWARE IS PROVIDED BY THE COPYRIGHT HOLDERS AND CONTRIBUTORS
   "AS IS" AND ANY EXPRESS OR IMPLIED WARRANTIES, INCLUDING, BUT NOT LIMITED
   TO, THE IMPLIED WARRANTIES OF MERCHANTABILITY AND FITNESS FOR A PARTICULAR
   PURPOSE ARE DISCLAIMED. IN NO EVENT SHALL THE COPYRIGHT HOLDER OR
   CONTRIBUTORS BE LIABLE FOR ANY DIRECT, INDIRECT, INCIDENTAL, SPECIAL,
   EXEMPLARY, OR CONSEQUENTIAL DAMAGES (INCLUDING, BUT NOT LIMITED TO,
   PROCUREMENT OF SUBSTITUTE GOODS OR SERVICES; LOSS OF USE, DATA, OR PROFITS;
   OR BUSINESS INTERRUPTION) HOWEVER CAUSED AND ON ANY THEORY OF LIABILITY,
   WHETHER IN CONTRACT, STRICT LIABILITY, OR TORT (INCLUDING NEGLIGENCE OR
   OTHERWISE) ARISING IN ANY WAY OUT OF THE USE OF THIS SOFTWARE, EVEN IF
   ADVISED OF THE POSSIBILITY OF SUCH DAMAGE.
   ----------------------------------------------------------------------------

   with the extension:

   You may distribute or publicly perform any modification only under the
   terms of this license.
   (Note, this means that if you distribute a modified file,
    the modified file must also be provided under this license).
*/

#ifdef __cplusplus
extern "C" {
#endif

#include "fmi2TypesPlatform.h"
#include "fmi2FunctionTypes.h"
#include <stdlib.h>

/*
  Export FMI2 API functions on Windows and under GCC.
  If custom linking is desired then the FMI2_Export must be
  defined before including this file. For instance,
  it may be set to __declspec(dllimport).
*/
#if !defined(FMI2_Export)
  #if !defined(FMI2_FUNCTION_PREFIX)
    #if defined _WIN32 || defined __CYGWIN__
     /* Note: both gcc & MSVC on Windows support this syntax. */
        #define FMI2_Export __declspec(dllexport)
    #else
      #if __GNUC__ >= 4
        #define FMI2_Export __attribute__ ((visibility ("default")))
      #else
        #define FMI2_Export
      #endif
    #endif
  #else
    #define FMI2_Export
  #endif
#endif

/* Macros to construct the real function name
   (prepend function name by FMI2_FUNCTION_PREFIX) */
#if defined(FMI2_FUNCTION_PREFIX)
  #define fmi2Paste(a,b)     a ## b
  #define fmi2PasteB(a,b)    fmi2Paste(a,b)
  #define fmi2FullName(name) fmi2PasteB(FMI2_FUNCTION_PREFIX, name)
#else
  #define fmi2FullName(name) name
#endif

/***************************************************
Common Functions
****************************************************/
#define fmi2GetTypesPlatform         fmi2FullName(fmi2GetTypesPlatform)
#define fmi2GetVersion               fmi2FullName(fmi2GetVersion)
#define fmi2SetDebugLogging          fmi2FullName(fmi2SetDebugLogging)
#define fmi2Instantiate              fmi2FullName(fmi2Instantiate)
#define fmi2FreeInstance             fmi2FullName(fmi2FreeInstance)
#define fmi2SetupExperiment          fmi2FullName(fmi2SetupExperiment)
#define fmi2EnterInitializationMode  fmi2FullName(fmi2EnterInitializationMode)
#define fmi2ExitInitializationMode   fmi2FullName(fmi2ExitInitializationMode)
#define fmi2Terminate                fmi2FullName(fmi2Terminate)
#define fmi2Reset                    fmi2FullName(fmi2Reset)
#define fmi2GetReal                  fmi2FullName(fmi2GetReal)
#define fmi2GetInteger               fmi2FullName(fmi2GetInteger)
#define fmi2GetBoolean               fmi2FullName(fmi2GetBoolean)
#define fmi2GetString                fmi2FullName(fmi2GetString)
#define fmi2SetReal                  fmi2FullName(fmi2SetReal)
#define fmi2SetInteger               fmi2FullName(fmi2SetInteger)
#define fmi2SetBoolean               fmi2FullName(fmi2SetBoolean)
#define fmi2SetString                fmi2FullName(fmi2SetString)
#define fmi2GetFMUstate              fmi2FullName(fmi2GetFMUstate)
#define fmi2SetFMUstate              fmi2FullName(fmi2SetFMUstate)
#define fmi2FreeFMUstate             fmi2FullName(fmi2FreeFMUstate)
#define fmi2SerializedFMUstateSize   fmi2FullName(fmi2SerializedFMUstateSize)
#define fmi2SerializeFMUstate        fmi2FullName(fmi2SerializeFMUstate)
#define fmi2DeSerializeFMUstate      fmi2FullName(fmi2DeSerializeFMUstate)
#define fmi2GetDirectionalDerivative fmi2FullName(fmi2GetDirectionalDerivative)

/***************************************************
Functions for FMI2 for Model Exchange
****************************************************/
#define fmi2EnterEventMode                fmi2FullName(fmi2EnterEventMode)
#define fmi2NewDiscreteStates             fmi2FullName(fmi2NewDiscreteStates)
#define fmi2EnterContinuousTimeMode       fmi2FullName(fmi2EnterContinuousTimeMode)
#define fmi2CompletedIntegratorStep       fmi2FullName(fmi2CompletedIntegratorStep)
#define fmi2SetTime                       fmi2FullName(fmi2SetTime)
#define fmi2SetContinuousStates           fmi2FullName(fmi2SetContinuousStates)
#define fmi2GetDerivatives                fmi2FullName(fmi2GetDerivatives)
#define fmi2GetEventIndicators            fmi2FullName(fmi2GetEventIndicators)
#define fmi2GetContinuousStates           fmi2FullName(fmi2GetContinuousStates)
#define fmi2GetNominalsOfContinuousStates fmi2FullName(fmi2GetNominalsOfContinuousStates)

/***************************************************
Functions for FMI2 for Co-Simulation
****************************************************/
#define fmi2SetRealInputDerivatives      fmi2FullName(fmi2SetRealInputDerivatives)
#define fmi2GetRealOutputDerivatives     fmi2FullName(fmi2GetRealOutputDerivatives)
#define fmi2DoStep                       fmi2FullName(fmi2DoStep)
#define fmi2CancelStep                   fmi2FullName(fmi2CancelStep)
#define fmi2GetStatus                    fmi2FullName(fmi2GetStatus)
#define fmi2GetRealStatus                fmi2FullName(fmi2GetRealStatus)
#define fmi2GetIntegerStatus             fmi2FullName(fmi2GetIntegerStatus)
#define fmi2GetBooleanStatus             fmi2FullName(fmi2GetBooleanStatus)
#define fmi2GetStringStatus              fmi2FullName(fmi2GetStringStatus)

/* Version number */
#define fmi2Version "2.0"

/***************************************************
Common Functions
****************************************************/

/* Inquire version numbers of header files */
   FMI2_Export fmi2GetTypesPlatformTYPE fmi2GetTypesPlatform;
   FMI2_Export fmi2GetVersionTYPE       fmi2GetVersion;
   FMI2_Export fmi2SetDebugLoggingTYPE  fmi2SetDebugLogging;

/* Creation and destruction of FMU instances */
   FMI2_Export fmi2InstantiateTYPE  fmi2Instantiate;
   FMI2_Export fmi2FreeInstanceTYPE fmi2FreeInstance;

/* Enter and exit initialization mode, terminate and reset */
   FMI2_Export fmi2SetupExperimentTYPE         fmi2SetupExperiment;
   FMI2_Export fmi2EnterInitializationModeTYPE fmi2EnterInitializationMode;
   FMI2_Export fmi2ExitInitializationModeTYPE  fmi2ExitInitializationMode;
   FMI2_Export fmi2TerminateTYPE               fmi2Terminate;
   FMI2_Export fmi2ResetTYPE                   fmi2Reset;

/* Getting and setting variables values */
   FMI2_Export fmi2GetRealTYPE    fmi2GetReal;
   FMI2_Export fmi2GetIntegerTYPE fmi2GetInteger;
   FMI2_Export fmi2GetBooleanTYPE fmi2GetBoolean;
   FMI2_Export fmi2GetStringTYPE  fmi2GetString;

   FMI2_Export fmi2SetRealTYPE    fmi2SetReal;
   FMI2_Export fmi2SetIntegerTYPE fmi2SetInteger;
   FMI2_Export fmi2SetBooleanTYPE fmi2SetBoolean;
   FMI2_Export fmi2SetStringTYPE  fmi2SetString;

/* Getting and setting the internal FMU state */
   FMI2_Export fmi2GetFMUstateTYPE            fmi2GetFMUstate;
   FMI2_Export fmi2SetFMUstateTYPE            fmi2SetFMUstate;
   FMI2_Export fmi2FreeFMUstateTYPE           fmi2FreeFMUstate;
   FMI2_Export fmi2SerializedFMUstateSizeTYPE fmi2SerializedFMUstateSize;
   FMI2_Export fmi2SerializeFMUstateTYPE      fmi2SerializeFMUstate;
   FMI2_Export fmi2DeSerializeFMUstateTYPE    fmi2DeSerializeFMUstate;

/* Getting partial derivatives */
   FMI2_Export fmi2GetDirectionalDerivativeTYPE fmi2GetDirectionalDerivative;

/***************************************************
Functions for FMI2 for Model Exchange
****************************************************/

/* Enter and exit the different modes */
   FMI2_Export fmi2EnterEventModeTYPE               fmi2EnterEventMode;
   FMI2_Export fmi2NewDiscreteStatesTYPE            fmi2NewDiscreteStates;
   FMI2_Export fmi2EnterContinuousTimeModeTYPE      fmi2EnterContinuousTimeMode;
   FMI2_Export fmi2CompletedIntegratorStepTYPE      fmi2CompletedIntegratorStep;

/* Providing independent variables and re-initialization of caching */
   FMI2_Export fmi2SetTimeTYPE             fmi2SetTime;
   FMI2_Export fmi2SetContinuousStatesTYPE fmi2SetContinuousStates;

/* Evaluation of the model equations */
   FMI2_Export fmi2GetDerivativesTYPE                fmi2GetDerivatives;
   FMI2_Export fmi2GetEventIndicatorsTYPE            fmi2GetEventIndicators;
   FMI2_Export fmi2GetContinuousStatesTYPE           fmi2GetContinuousStates;
   FMI2_Export fmi2GetNominalsOfContinuousStatesTYPE fmi2GetNominalsOfContinuousStates;

/***************************************************
Functions for FMI2 for Co-Simulation
****************************************************/

/* Simulating the slave */
   FMI2_Export fmi2SetRealInputDerivativesTYPE  fmi2SetRealInputDerivatives;
   FMI2_Export fmi2GetRealOutputDerivativesTYPE fmi2GetRealOutputDerivatives;

   FMI2_Export fmi2DoStepTYPE     fmi2DoStep;
   FMI2_Export fmi2CancelStepTYPE fmi2CancelStep;

/* Inquire slave status */
   FMI2_Export fmi2GetStatusTYPE        fmi2GetStatus;
   FMI2_Export fmi2GetRealStatusTYPE    fmi2GetRealStatus;
   FMI2_Export fmi2GetIntegerStatusTYPE fmi2GetIntegerStatus;
   FMI2_Export fmi2GetBooleanStatusTYPE fmi2GetBooleanStatus;
   FMI2_Export fmi2GetStringStatusTYPE  fmi2GetStringStatus;

#ifdef __cplusplus
}  /* end of extern "C" { */
#endif

#endif /* fmi2Functions_h */
```

#### fmuTemplate.h
```c
/*****************************************************************************/
/* FILE fmi2Functions.h */
/*****************************************************************************/

#include <stdio.h>
#include <string.h>
#include <assert.h>

#include "fmi2Functions.h"

#define compEnv comp->functions.componentEnvironment
#define compLog comp->functions.logger

#define not_modelError (modelInstantiated | modelInitialized | modelTerminated)
/* According to the chart on pg. 85 of the spec, 'Get's are not allowed
	until after we enter initialization mode, so use validGet instead */
#define validGet (modelInitialized | modelTerminated)

typedef enum {
	modelInstantiated = 1<<0,
	modelInitialized  = 1<<1,
	modelTerminated   = 1<<2,
	modelError        = 1<<3
} ModelState;

typedef struct {
	SolverStruct			S;
	fmi2Boolean				*b;
	fmi2String				*s;
	fmi2String				instanceName;
	fmi2String				GUID;
	fmi2Type					fmuType;
	fmi2CallbackFunctions	functions;
	fmi2Boolean				loggingOn;
	fmi2Boolean				synced;
	fmi2Boolean				jsynced;
	ModelState				state;
	fmi2Real				*Jacobian;
	fmi2Real				*initRes;
	fmi2Real				*initJacobian;

	fmi2Real				tolerance;
	fmi2Real				startTime;
	fmi2Boolean				stopTimeDefined;
	fmi2Real				stopTime;
	fmi2Real				lastStepSize;

	fmi2Real				lastEventTime;
	fmi2Real				lastSuccessfulTime;

	fmi2Boolean				initializeMode;
	FILE					*fptr;
	fmi2String				fstr;
	fmi2Integer				numpts;
	fmi2Real				lastsampletime;
	fmi2Real				minSampleStep;

	fmi2Integer				vidsts; /* -1 = error, 0 = no data, 1 = init, 2 = int */
	fmi2Char				viderror[MAXERRSTRLENGTH+1];
	fmi2Real				vidlasttime;
} ModelInstance;
```
